FUNCTION_BLOCK EL1512
VAR
	_io : EL1512_Data;
	{attribute addProperty Name "WcState"}
	_wcState : WcStateInputToggle;
	{attribute addProperty Name "Info data"}
	_infoData : InfoDataAds;
END_VAR

PROPERTY IO : REFERENCE TO EL1512_Data
GET
IO REF= _io;
END_GET
END_PROPERTY

PROPERTY WcState : REFERENCE TO WcStateInputToggle
GET
WcState REF= _wcState;
END_GET
END_PROPERTY

END_FUNCTION_BLOCK

(* stored: Version 1.1.0.1, ProductVersion 3.1.4024.9
   POU EL1512: Id {8ac0c417-629f-0746-1984-7fe01d85ce68}, SpecialFunc None
   Property IO: Id {21f49c6a-45ef-0a24-0527-f57c167bafc5}
   Get Get: Id {eaebc8df-0571-03dc-3ee5-2d8cd2e52a59}
   Property WcState: Id {81a43219-6773-0953-10c9-32481fa73fc0}
   Get Get: Id {5ef978a2-ea56-0a69-2e33-b853f7f6231e} *)
